// TwinCAT 3 PLC project TcoPneumatics
// Title: TcoPneumatics
// Company: Vortex.Library
// Author: Dustin Hullett
// ProjectVersion: 0.6.0.913
// ProgramVersion: 3.1.4024.12
// libraries:
//   Tc2_Standard, * (Beckhoff Automation GmbH)
//   Tc2_System, * (Beckhoff Automation GmbH)
//   Tc3_Module, * (Beckhoff Automation GmbH)
//   TcoCore, 0.6.0.913 (Vortex.Library)
// project tree:
//   POUs/Cylinders/Base/ TcoCylinderBase.TcPOU, TcoDoubleCylinderBase.TcPOU
//   POUs/Cylinders/ TcoCylinder.TcPOU, TcoCylinderConfig.TcDUT, TcoCylinderStatus.TcDUT, TcoCylinderMoveTask.TcPOU, ITcoCylinder.TcIO, TcoDoubleCylinder.TcPOU
//   Version/ Global_Version.TcGVL
// real-time tasks:
//   TASK PlcTask: cycle T#10ms, priority 20, ADS port 350
//   TASK PlcTask1: cycle T#10ms, priority 21, ADS port 351

// ---- POUs/Cylinders/TcoCylinderConfig.TcDUT
TYPE TcoCylinderConfig :
STRUCT
    TimeToReachHomePosition : TIME := T#10S;
    TimeToReachWorkPosition : TIME := T#10S;
    TimeToRefill : TIME := T#1000MS;
END_STRUCT
END_TYPE

// ---- POUs/Cylinders/TcoCylinderStatus.TcDUT
TYPE TcoCylinderStatus :
STRUCT
    ActionDescription : STRING(100);
END_STRUCT
END_TYPE

// ---- Version/Global_Version.TcGVL
{attribute 'TcGenerated'}
{attribute 'no-analysis'}
{attribute 'linkalways'}
// This function has been automatically generated from the project information.
VAR_GLOBAL CONSTANT
    {attribute 'const_non_replaced'}
    stLibVersion_TcoPneumatics : ST_LibVersion := (
        iMajor := 0,
        iMinor := 1,
        iBuild := 0,
        iRevision := 54,
        nFlags := 0,
        sVersion := '0.1.0.54');
END_VAR

// ---- POUs/Cylinders/ITcoCylinder.TcIO
INTERFACE ITcoCylinder EXTENDS __System.IQueryInterface

PROPERTY AtHome : bool
GET
END_GET
END_PROPERTY

PROPERTY AtWork : bool
GET
END_GET
END_PROPERTY

METHOD MoveToHome : TcoCore.ITcoTaskStatus
END_METHOD

METHOD MoveToWork :TcoCore.ITcoTaskStatus
END_METHOD

(*~
	<docu>
		<summary>
			Stops cyclinder movement.
		 	<remarks>
				<note type="important">
					This method switched off the signals for the movement of the piston in both direction.
					However depending on the pnemumatics configuration the movement may contintue if designed in that way.
					THIS IS NOT A SAFETY FUCTION!
				</note>
			</remarks>
		</summary>
	</docu>
~*)
METHOD Stop : TcoCore.ITcoTaskStatus
END_METHOD

END_INTERFACE

// ---- POUs/Cylinders/Base/TcoCylinderBase.TcPOU
FUNCTION_BLOCK ABSTRACT TcoCylinderBase EXTENDS TcoCore.TcoComponent IMPLEMENTS ITcoCylinder
VAR_IN_OUT
    (*~
        <docu>
            <summary>
                Home position sensor.
            </summary>
        </docu>
    ~*)
    {attribute addProperty Name "<#Home position sensor#>"}
    inoAtHomePos : BOOL;
    (*~
        <docu>
            <summary>
                Working position sensor.
            </summary>
        </docu>
    ~*)
    {attribute addProperty Name "<#Work position sensor#>"}
    inoAtWorkPos : BOOL;
END_VAR
VAR_IN_OUT
    (*~
        <docu>
            <summary>
                Move to working home position signal.
            </summary>
        </docu>
    ~*)
    {attribute addProperty Name "<#Move to home position actuator#>"}
    inoToHomePos : BOOL;
    (*~
        <docu>
            <summary>
                Move to working posistion signal.
            </summary>
        </docu>
    ~*)
    {attribute addProperty Name "<#Move to work position actuator#>"}
    inoToWorkPos : BOOL;
END_VAR
VAR
    (*~
        <docu>
            <summary>
                Home position sensor.
            </summary>
        </docu>
    ~*)
    {attribute addProperty Name "<#Home position sensor#>"}
    _atHomePos : BOOL;
    (*~
        <docu>
            <summary>
                Working position sensor.
            </summary>
        </docu>
    ~*)
    {attribute addProperty Name "<#Work position sensor#>"}
    _atWorkPos : BOOL;
    (*~
        <docu>
            <summary>
                Move to working home position signal.
            </summary>
        </docu>
    ~*)
    {attribute addProperty Name "<#Move to home position actuator#>"}
    _toHomePos : BOOL;
    (*~
        <docu>
            <summary>
                Move to working posistion signal.
            </summary>
        </docu>
    ~*)
    {attribute addProperty Name "<#Move to work position actuator#>"}
    _toWorkPos : BOOL;
END_VAR
VAR
    {attribute addProperty Name "<#Home sensor signal#>"}
    _atHomePosSignalInfo : TcoCore.TcoSignalInfo;
    {attribute addProperty Name "<#Work sensor signal#>"}
    _atWorkPosSignalInfo : TcoCore.TcoSignalInfo;
    {attribute addProperty Name "<#Move to home position signal#>"}
    _toHomePosSignalInfo : TcoCore.TcoSignalInfo;
    {attribute addProperty Name "<#Move to work position signal#>"}
    _toWorkPosSignalInfo : TcoCore.TcoSignalInfo;
END_VAR

IF (__ISVALIDREF(inoAtHomePos)) THEN
    _atHomePos := inoAtHomePos;
    _atHomePosSignalInfo.GetSignalInfo(SIZEOF(inoAtHomePos), ADR(inoAtHomePos));
END_IF;

IF (__ISVALIDREF(inoAtWorkPos)) THEN
    _atWorkPos := inoAtWorkPos;
    _atWorkPosSignalInfo.GetSignalInfo(SIZEOF(inoAtWorkPos), ADR(inoAtWorkPos));
END_IF;

IF (__ISVALIDREF(inoToHomePos)) THEN
    inoToHomePos := _toHomePos;
    _toHomePosSignalInfo.GetSignalInfo(SIZEOF(inoToHomePos), ADR(inoToHomePos));
END_IF;

IF (__ISVALIDREF(inoToWorkPos)) THEN
    inoToWorkPos := _toWorkPos;
    _toWorkPosSignalInfo.GetSignalInfo(SIZEOF(inoToWorkPos), ADR(inoToWorkPos));
END_IF;

(*~
    <docu>
        <summary>
            Gets whether the piston is in home position.
        </summary>
    </docu>
~*)
PROPERTY AtHome : bool
GET
AtHome := THIS^._atHomePos;
END_GET
END_PROPERTY

(*~
    <docu>
        <summary>
            Gets whether the piston is in work position.
        </summary>
    </docu>
~*)
PROPERTY AtWork : bool
GET
AtWork := _atWorkPos;
END_GET
END_PROPERTY

METHOD FB_init : BOOL
VAR_INPUT
    bInitRetains : BOOL; // if TRUE, the retain variables are initialized (warm start / cold start)
    bInCopyCode : BOOL; // if TRUE, the instance afterwards gets moved into the copy code (online change)
    ParentObject : ITcoObject;
END_VAR
END_METHOD

(*~
    <docu>
        <summary>
            Gets the `MoveHomeTask` task that controls the moving of the cyclinder in home position.
            <remarks>
                <note type="important">
                    This is an abstract method and must be implemented in derived class.
                </note>
            </remarks>
        </summary>
    </docu>
~*)
PROPERTY PUBLIC ABSTRACT MoveHomeTask : TcoCore.ITcoTask
GET
END_GET
END_PROPERTY

(*~
    <docu>
        <summary>
            Starts movement into home position.
        </summary>
    </docu>
~*)
METHOD MoveToHome : TcoCore.ITcoTaskStatus
IF (MoveHomeTask <> 0) THEN
    MoveToHome := MoveHomeTask.Invoke();
END_IF;
END_METHOD

(*~
    <docu>
        <summary>
            Starts movement into work position.
        </summary>
    </docu>
~*)
METHOD MoveToWork : TcoCore.ITcoTaskStatus
IF (MoveWorkTask <> 0) THEN
    MoveToWork := MoveWorkTask.Invoke();
END_IF;
END_METHOD

(*~
    <docu>
        <summary>
            Gets the `MoveWorkTask` task that controls the moving of the cyclinder into work position.
            <remarks>
                <note type="important">
                    This is an abstract method and must be implemented in derived class.
                </note>
            </remarks>
        </summary>
    </docu>
~*)
PROPERTY PUBLIC ABSTRACT MoveWorkTask : TcoCore.ITcoTask
GET
END_GET
END_PROPERTY

(*~
    <docu>
        <summary>
            Restore all tasks of this instance into initial state.
        </summary>
    </docu>
~*)
METHOD Restore : ITcoRestorable
IF (MoveHomeTask <> 0) THEN
    MoveHomeTask.Restore();
END_IF;

IF (MoveWorkTask <> 0) THEN
    MoveWorkTask.Restore();
END_IF;

IF (StopTask <> 0) THEN
    StopTask.Restore();
END_IF;
END_METHOD

METHOD PROTECTED ServiceMode
END_METHOD

(*~
    <docu>
        <summary>
            Stops cyclinder movement.
             <remarks>
                <note type="important">
                    This method switched off the signals for the movement of the piston in both direction.
                    However depending on the pnemumatics configuration the movement may contintue if designed in that way.
                    THIS IS NOT A SAFETY FUCTION!
                </note>
            </remarks>
        </summary>
    </docu>
~*)
METHOD Stop : TcoCore.ITcoTaskStatus
IF (StopTask <> 0) THEN
    Stop := StopTask.Invoke();
END_IF;
END_METHOD

(*~
    <docu>
        <summary>
            Gets the `StopTask` task that controls the stopping cyclinder movement.
            <remarks>
                <note type="important">
                    This is an abstract method and must be implemented in derived class.
                </note>
            </remarks>
        </summary>
    </docu>
~*)
PROPERTY PUBLIC ABSTRACT StopTask : TcoCore.ITcoTask
GET
END_GET
END_PROPERTY

END_FUNCTION_BLOCK

// ---- POUs/Cylinders/Base/TcoDoubleCylinderBase.TcPOU
FUNCTION_BLOCK ABSTRACT TcoDoubleCylinderBase EXTENDS TcoCore.TcoComponent IMPLEMENTS ITcoCylinder
VAR_IN_OUT
    (*~
        <docu>
            <summary>
                Home position sensor 1.
            </summary>
        </docu>
    ~*)
    {attribute addProperty Name "<#Home position sensor#> - 1"}
    inoAtHomePos1 : BOOL;
    (*~
        <docu>
            <summary>
                Home position sensor 2.
            </summary>
        </docu>
    ~*)
    {attribute addProperty Name "<#Home position sensor#> - 2"}
    inoAtHomePos2 : BOOL;
    (*~
        <docu>
            <summary>
                Working position sensor 1.
            </summary>
        </docu>
    ~*)
    {attribute addProperty Name "<#Work position sensor#> - 1"}
    inoAtWorkPos1 : BOOL;
    (*~
        <docu>
            <summary>
                Working position sensor 1.
            </summary>
        </docu>
    ~*)
    {attribute addProperty Name "<#Work position sensor#> - 2"}
    inoAtWorkPos2 : BOOL;
END_VAR
VAR_IN_OUT
    (*~
        <docu>
            <summary>
                Move to working home position signal.
            </summary>
        </docu>
    ~*)
    {attribute addProperty Name "<#Move to home position actuator#>"}
    inoToHomePos : BOOL;
    (*~
        <docu>
            <summary>
                Move to working posistion signal.
            </summary>
        </docu>
    ~*)
    {attribute addProperty Name "<#Move to work position actuator#>"}
    inoToWorkPos : BOOL;
END_VAR
VAR
    (*~
        <docu>
            <summary>
                Home position sensor.
            </summary>
        </docu>
    ~*)
    {attribute addProperty Name "<#Home position sensor#>"}
    _atHomePos : BOOL;
    (*~
        <docu>
            <summary>
                Working position sensor.
            </summary>
        </docu>
    ~*)
    {attribute addProperty Name "<#Work position sensor#>"}
    _atWorkPos : BOOL;
    (*~
        <docu>
            <summary>
                Move to working home position signal.
            </summary>
        </docu>
    ~*)
    {attribute addProperty Name "<#Move to home position actuator#>"}
    _toHomePos : BOOL;
    (*~
        <docu>
            <summary>
                Move to working posistion signal.
            </summary>
        </docu>
    ~*)
    {attribute addProperty Name "<#Move to work position actuator#>"}
    _toWorkPos : BOOL;
END_VAR
VAR
    {attribute addProperty Name "<#Home sensor signal 1#>"}
    _atHomePos1SignalInfo : TcoCore.TcoSignalInfo;
    {attribute addProperty Name "<#Home sensor signal 2#>"}
    _atHomePos2SignalInfo : TcoCore.TcoSignalInfo;
    {attribute addProperty Name "<#Work sensor signal 1#>"}
    _atWorkPos1SignalInfo : TcoCore.TcoSignalInfo;
    {attribute addProperty Name "<#Work sensor signal 2#>"}
    _atWorkPos2SignalInfo : TcoCore.TcoSignalInfo;
    {attribute addProperty Name "<#Move to home position signal#>"}
    _toHomePosSignalInfo : TcoCore.TcoSignalInfo;
    {attribute addProperty Name "<#Move to work position signal#>"}
    _toWorkPosSignalInfo : TcoCore.TcoSignalInfo;
END_VAR

IF (__ISVALIDREF(inoAtHomePos1) AND __ISVALIDREF(inoAtHomePos2)) THEN
    _atHomePos := inoAtHomePos1 AND inoAtHomePos2;
    _atHomePos1SignalInfo.GetSignalInfo(SIZEOF(inoAtHomePos1), ADR(inoAtHomePos1));
    _atHomePos2SignalInfo.GetSignalInfo(SIZEOF(inoAtHomePos2), ADR(inoAtHomePos2));
END_IF;

IF (__ISVALIDREF(inoAtWorkPos1) AND __ISVALIDREF(inoAtWorkPos2)) THEN
    _atWorkPos := inoAtWorkPos1 AND inoAtWorkPos2;
    _atWorkPos1SignalInfo.GetSignalInfo(SIZEOF(inoAtWorkPos1), ADR(inoAtWorkPos1));
    _atWorkPos2SignalInfo.GetSignalInfo(SIZEOF(inoAtWorkPos2), ADR(inoAtWorkPos2));
END_IF;

IF (__ISVALIDREF(inoToHomePos)) THEN
    inoToHomePos := _toHomePos;
    _toHomePosSignalInfo.GetSignalInfo(SIZEOF(inoToHomePos), ADR(inoToHomePos));
END_IF;

IF (__ISVALIDREF(inoToWorkPos)) THEN
    inoToWorkPos := _toWorkPos;
    _toWorkPosSignalInfo.GetSignalInfo(SIZEOF(inoToWorkPos), ADR(inoToWorkPos));
END_IF;

(*~
    <docu>
        <summary>
            Gets whether the piston is in home position.
        </summary>
    </docu>
~*)
PROPERTY AtHome : bool
GET
AtHome := THIS^._atHomePos;
END_GET
END_PROPERTY

(*~
    <docu>
        <summary>
            Gets whether the piston is in work position.
        </summary>
    </docu>
~*)
PROPERTY AtWork : bool
GET
AtWork := _atWorkPos;
END_GET
END_PROPERTY

METHOD FB_init : BOOL
VAR_INPUT
    bInitRetains : BOOL; // if TRUE, the retain variables are initialized (warm start / cold start)
    bInCopyCode : BOOL; // if TRUE, the instance afterwards gets moved into the copy code (online change)
    ParentObject : ITcoObject;
END_VAR
END_METHOD

(*~
    <docu>
        <summary>
            Gets the `MoveHomeTask` task that controls the moving of the cyclinder in home position.
            <remarks>
                <note type="important">
                    This is an abstract method and must be implemented in derived class.
                </note>
            </remarks>
        </summary>
    </docu>
~*)
PROPERTY PUBLIC ABSTRACT MoveHomeTask : TcoCore.ITcoTask
GET
END_GET
END_PROPERTY

(*~
    <docu>
        <summary>
            Starts movement into home position.
        </summary>
    </docu>
~*)
METHOD MoveToHome : TcoCore.ITcoTaskStatus
IF (MoveHomeTask <> 0) THEN
    MoveToHome := MoveHomeTask.Invoke();
END_IF;
END_METHOD

(*~
    <docu>
        <summary>
            Starts movement into work position.
        </summary>
    </docu>
~*)
METHOD MoveToWork : TcoCore.ITcoTaskStatus
IF (MoveWorkTask <> 0) THEN
    MoveToWork := MoveWorkTask.Invoke();
END_IF;
END_METHOD

(*~
    <docu>
        <summary>
            Gets the `MoveWorkTask` task that controls the moving of the cyclinder into work position.
            <remarks>
                <note type="important">
                    This is an abstract method and must be implemented in derived class.
                </note>
            </remarks>
        </summary>
    </docu>
~*)
PROPERTY PUBLIC ABSTRACT MoveWorkTask : TcoCore.ITcoTask
GET
END_GET
END_PROPERTY

(*~
    <docu>
        <summary>
            Restore all tasks of this instance into initial state.
        </summary>
    </docu>
~*)
METHOD Restore : ITcoRestorable
IF (MoveHomeTask <> 0) THEN
    MoveHomeTask.Restore();
END_IF;

IF (MoveWorkTask <> 0) THEN
    MoveWorkTask.Restore();
END_IF;

IF (StopTask <> 0) THEN
    StopTask.Restore();
END_IF;
END_METHOD

METHOD PROTECTED ServiceMode
END_METHOD

(*~
    <docu>
        <summary>
            Stops cyclinder movement.
             <remarks>
                <note type="important">
                    This method switched off the signals for the movement of the piston in both direction.
                    However depending on the pnemumatics configuration the movement may contintue if designed in that way.
                    THIS IS NOT A SAFETY FUCTION!
                </note>
            </remarks>
        </summary>
    </docu>
~*)
METHOD Stop : TcoCore.ITcoTaskStatus
IF (StopTask <> 0) THEN
    Stop := StopTask.Invoke();
END_IF;
END_METHOD

(*~
    <docu>
        <summary>
            Gets the `StopTask` task that controls the stopping cyclinder movement.
            <remarks>
                <note type="important">
                    This is an abstract method and must be implemented in derived class.
                </note>
            </remarks>
        </summary>
    </docu>
~*)
PROPERTY PUBLIC ABSTRACT StopTask : TcoCore.ITcoTask
GET
END_GET
END_PROPERTY

END_FUNCTION_BLOCK

// ---- POUs/Cylinders/TcoCylinder.TcPOU
{attribute addProperty _moveHomeDefaultName "<#MOVE HOME#>"}
{attribute addProperty _moveWorkDefaultName "<#MOVE TO WORK#>"}
{attribute addProperty _stopDefaultName "<#STOP#>"}
FUNCTION_BLOCK TcoCylinder EXTENDS TcoCylinderBase
VAR
    {attribute addProperty Name "|[[1]Attribute_moveHomeDefaultName]|"}
    _moveHomeDefault : TcoCylinderMoveTask(THIS^);
    {attribute addProperty Name "|[[1]Attribute_moveWorkDefaultName]|"}
    _moveWorkDefault : TcoCylinderMoveTask(THIS^);
    {attribute addProperty Name "|[[1]Attribute_stopDefaultName]|"}
    _stopDefault : TcoCore.TcoTask(THIS^);
	increment: INT;
	_suspendedHome:BOOL;
	_suspendedWork:BOOL;
	{attribute 'hide'} 
	_suspendedHomeCounter:INT;
	{attribute 'hide'} 
	_suspendedWorkCounter:INT;
END_VAR
VAR
    _config : TcoCylinderConfig;
	_status : TcoCylinderStatus;
	_refillTimer:TON;	
END_VAR

SUPER^(inoAtHomePos := inoAtHomePos, inoAtWorkPos := inoAtWorkPos, inoToHomePos := inoToHomePos, inoToWorkPos := inoToWorkPos);
_suspendedHomeCounter:=0;
_suspendedWorkCounter:=0;

	
IF(_atHomePos AND _atWorkPos) THEN Messenger.Error('<#Home and work position sensors are both active. Check the position of sensors!#>'); END_IF;

// Disables mutualy exclusive actions
_moveWorkDefault.Enabled := TRUE;// NOT _moveHomeDefault.Busy;


_moveHomeDefault(PositionSensor := _atHomePos AND NOT _atWorkPos,
    MoveToPositionSignal := _toHomePos,
    InverseSignal := _toWorkPos,
	TimeToRefill:=_config.TimeToRefill,
	refInverseTask:=_moveWorkDefault,
    MaxTimeToReachPosition := _config.TimeToReachHomePosition,
    PositionName := '<#Home#>');


	
// Disables mutualy exclusive actions		
_moveHomeDefault.Enabled := TRUE;//NOT _moveWorkDefault.Busy;
	
_moveWorkDefault(PositionSensor := _atWorkPos AND NOT _atHomePos,
    MoveToPositionSignal := _toWorkPos,
    InverseSignal := _toHomePos,
	TimeToRefill:=_config.TimeToRefill,
	refInverseTask:=_moveHomeDefault,
    MaxTimeToReachPosition := _config.TimeToReachWorkPosition,
    PositionName := '<#Work#>');
	

IF (_stopDefault.Execute()) THEN
	_toHomePos := FALSE;
	_toWorkPos := FALSE;
    _moveHomeDefault.Abort();
    _moveWorkDefault.Abort();
    _stopDefault.Abort();
    _moveHomeDefault.Restore();
    _moveWorkDefault.Restore();
    _stopDefault.Restore();
    _stopDefault.DoneWhen(TRUE);
END_IF



// For further discussion about Status
IF(_moveHomeDefault.Busy) THEN
	_status.ActionDescription := 'Moving to home position';
ELSIF(_moveWorkDefault.Busy) THEN
	_status.ActionDescription := 'Moving to work position';
ELSIF(_stopDefault.Busy) THEN
	_status.ActionDescription := 'Stopping pressure';
ELSE	
	_status.ActionDescription := 'Idle';
END_IF

SUPER^(inoAtHomePos := inoAtHomePos, inoAtWorkPos := inoAtWorkPos, inoToHomePos := inoToHomePos, inoToWorkPos := inoToWorkPos);

(*~
	<docu>
		<summary>
			Aborts the movement to home position when the condition is 'true'.
		</summary>
		<remarks>			
				<note type="warning">
					The call of this method will be effective only when called AFTER the initialization of the instance of given TcoCylinder.
				</note>
		</remarks>	
	</docu>
~*)
METHOD AbortMoveHome : BOOL
VAR_IN_OUT
	(*~
	<docu>
		<summary>
			Condition to abort the movement of the cylinder.
		</summary>	
	</docu>
	~*)
	inoDisableCondition : BOOL;
END_VAR
VAR
	_signalInfo : TcoSignalInfo;
END_VAR
IF (_toHomePos OR _moveHomeDefault.Busy) AND inoDisableCondition THEN
	_signalInfo.GetSignalInfo(SIZEOF(inoDisableCondition), ADR(inoDisableCondition));
	Messenger.Build().Append('<#Movement aborted due to#> : ').Append(_signalInfo.SymbolPath).As().AsError().Pin();
	_toHomePos := FALSE;
	IF(__ISVALIDREF(THIS^.inoToHomePos)) THEN THIS^.inoToHomePos := FALSE; END_IF;
	_moveHomeDefault.Abort();
END_IF
END_METHOD

(*~
	<docu>
		<summary>
			Aborts the movement to work position when the condition is 'true'.
		</summary>
		<remarks>			
				<note type="warning">
					The call of this method will be effective only when called AFTER the initialization of the instance of given TcoCylinder.
				</note>
		</remarks>	
	</docu>
~*)
METHOD AbortMoveWork : BOOL
VAR_IN_OUT
	(*~
		<docu>
			<summary>
				Condition to abort the movement of the cylinder.
			</summary>	
		</docu>
	~*)
	inoDisableCondition : BOOL;
END_VAR
VAR
	_signalInfo : TcoSignalInfo;
END_VAR
IF (_toWorkPos OR _moveWorkDefault.Busy) AND inoDisableCondition THEN
	_signalInfo.GetSignalInfo(SIZEOF(inoDisableCondition), ADR(inoDisableCondition));
	Messenger.Build().Append('<#Movement aborted due to#> : ').Append(_signalInfo.SymbolPath).As().AsError().Pin();
	_toWorkPos := FALSE;
	IF(__ISVALIDREF(THIS^.inoToWorkPos)) THEN THIS^.inoToWorkPos := FALSE; END_IF;
	_moveWorkDefault.Abort();
END_IF
END_METHOD

(*~
	<docu>
		<summary>
			Gets the configuration of the cylinder. 					
		</summary>			
	</docu>	
~*)
PROPERTY Config : REFERENCE TO TcoCylinderConfig
GET
Config REF= _config;
END_GET
END_PROPERTY

(*~
	<docu>
		<summary>
			Gets the `MoveHomeTask` task that controls the moving of the cyclinder in home position. 		
		</summary>			
	</docu>	
~*)
PROPERTY MoveHomeTask : TcoCore.ITcoTask
GET
MoveHomeTask := _moveHomeDefault;
END_GET
END_PROPERTY

(*~
	<docu>
		<summary>
			Gets the `MoveWorkTask` task that controls the moving of the cyclinder into work position. 		
		</summary>			
	</docu>	
~*)
PROPERTY MoveWorkTask : TcoCore.ITcoTask
GET
MoveWorkTask := _moveWorkDefault;
END_GET
END_PROPERTY

(*~
	<docu>
		<summary>
			Refill cylinder after booth outputs are off .
		</summary>
		<remarks>			
				<note type="warning">
					The call of this method will be effective only when called AFTER the initialization of the instance of given TcoCylinder and methods like AbortMoveHone,SuspendMoveHom...
				</note>
		</remarks>	
	</docu>
~*)
METHOD Refill : BOOL
VAR_INPUT
	(*~
	<docu>
		<summary>
			Time of refill cylinder after aborting or suspending
		</summary>	
	</docu>
	~*)
	inRefillTime:TIME;
END_VAR

_refillTimer(In:=inoToHomePos XOR  inoToWorkPos ,Pt:=T#49D);

_config.TimeToRefill:=inRefillTime;

IF  _refillTimer.ET>T#0MS
	AND _refillTimer.ET<_config.TimeToRefill  
	AND _config.TimeToRefill<>T#0S THEN
	_toHomePos	 := TRUE;
	_toWorkPos	 := TRUE;	
END_IF;

	
SUPER^(inoAtHomePos := inoAtHomePos, inoAtWorkPos := inoAtWorkPos, inoToHomePos := inoToHomePos, inoToWorkPos := inoToWorkPos);
END_METHOD

PROPERTY Status : REFERENCE TO TcoCylinderStatus
GET
Status REF= _status;
END_GET
END_PROPERTY

(*~
	<docu>
		<summary>
			Gets the `StopTask` task that controls the stopping of the cyclinder. 		
		</summary>			
	</docu>	
~*)
PROPERTY StopTask : TcoCore.ITcoTask
GET
StopTask := _stopDefault;
END_GET
END_PROPERTY

(*~
	<docu>
		<summary>
			Suspend the movement to home position when the condition is 'true'. Task is still busy
		</summary>
		<remarks>			
				<note type="warning">
					The call of this method will be effective only when called AFTER the initialization of the instance of given TcoCylinder.
				</note>
		</remarks>	
	</docu>
~*)
METHOD SuspendMoveHome : BOOL
VAR_IN_OUT
	(*~
	<docu>
		<summary>
			Condition to abort the movement of the cylinder.
		</summary>	
	</docu>
	~*)
	inoDisableCondition : BOOL;
END_VAR
VAR
	_signalInfo : TcoSignalInfo;
END_VAR
IF inoDisableCondition THEN
	_suspendedHomeCounter:=_suspendedHomeCounter+1;
END_IF
_suspendedHome:=_suspendedHomeCounter>0;

IF (_toHomePos OR _moveHomeDefault.Busy) AND inoDisableCondition THEN
	_signalInfo.GetSignalInfo(SIZEOF(inoDisableCondition), ADR(inoDisableCondition));
	Messenger.Warning(CONCAT('<#Movement suspended due to#> : ' , _signalInfo.SymbolPath));
	_toHomePos := FALSE;
	IF(__ISVALIDREF(THIS^.inoToHomePos)) THEN THIS^.inoToHomePos := FALSE; END_IF;
	
END_IF
END_METHOD

METHOD SuspendMoveHomeExpression : BOOL
VAR_INPUT
		inDisableCondition : BOOL;
		inMessage:STRING;
END_VAR
IF inDisableCondition THEN
	_suspendedHomeCounter:=_suspendedHomeCounter+1;
END_IF
_suspendedHome:=_suspendedHomeCounter>0;

IF (_toHomePos OR _moveHomeDefault.Busy) AND inDisableCondition THEN
	Messenger.Warning(CONCAT('<#Movement suspended due to#> : ' , inMessage));
	_toHomePos := FALSE;
	IF(__ISVALIDREF(THIS^.inoToHomePos)) THEN THIS^.inoToHomePos := FALSE; END_IF;
	
END_IF;
END_METHOD

(*~
	<docu>
		<summary>
			Suspend the movement to home position when the condition is NOT 'true'. Task is still busy
		</summary>
		<remarks>			
				<note type="warning">
					The call of this method will be effective only when called AFTER the initialization of the instance of given TcoCylinder.
				</note>
		</remarks>	
	</docu>
~*)
METHOD SuspendMoveHomeInverted : BOOL
VAR_IN_OUT
	(*~
	<docu>
		<summary>
			Condition to abort the movement of the cylinder.
		</summary>	
	</docu>
	~*)
	inoDisableCondition : BOOL;
END_VAR
VAR
	_signalInfo : TcoSignalInfo;
END_VAR
IF inoDisableCondition THEN
	_suspendedHomeCounter:=_suspendedHomeCounter+1;
END_IF
_suspendedHome:=_suspendedHomeCounter>0;

IF (_toHomePos OR _moveHomeDefault.Busy) AND not inoDisableCondition THEN
	_signalInfo.GetSignalInfo(SIZEOF(inoDisableCondition), ADR(inoDisableCondition));
	Messenger.Warning(CONCAT('<#Movement suspended due to NOT#> : ' , _signalInfo.SymbolPath));
	_toHomePos := FALSE;
	IF(__ISVALIDREF(THIS^.inoToHomePos)) THEN THIS^.inoToHomePos := FALSE; END_IF;
	
END_IF
END_METHOD

(*~
	<docu>
		<summary>
			Suspend the movement to work position when the condition is 'true'. Task is still bussy
		</summary>
		<remarks>			
				<note type="warning">
					The call of this method will be effective only when called AFTER the initialization of the instance of given TcoCylinder.
				</note>
		</remarks>	
	</docu>
~*)
METHOD SuspendMoveWork : BOOL
VAR_IN_OUT
	(*~
		<docu>
			<summary>
				Condition to abort the movement of the cylinder.
			</summary>	
		</docu>
	~*)
	inoDisableCondition : BOOL;
END_VAR
VAR
	_signalInfo : TcoSignalInfo;
END_VAR
IF inoDisableCondition THEN
	_suspendedWorkCounter:=_suspendedWorkCounter+1;
END_IF
_suspendedWork:=_suspendedWorkCounter>0;

IF (_toWorkPos OR _moveWorkDefault.Busy) AND inoDisableCondition THEN
	_signalInfo.GetSignalInfo(SIZEOF(inoDisableCondition), ADR(inoDisableCondition));
	Messenger.Warning(CONCAT('<#Movement suspended due to#> : ' , _signalInfo.SymbolPath));
	_toWorkPos := FALSE;
	IF(__ISVALIDREF(THIS^.inoToWorkPos)) THEN THIS^.inoToWorkPos := FALSE; END_IF;

END_IF
END_METHOD

METHOD SuspendMoveWorkExpression : BOOL
VAR_INPUT
		inDisableCondition : BOOL;
		inMessage:STRING;
END_VAR
IF inDisableCondition THEN
	_suspendedWorkCounter:=_suspendedWorkCounter+1;
END_IF
_suspendedWork:=_suspendedWorkCounter>0;

IF (_toWorkPos OR _moveWorkDefault.Busy) AND inDisableCondition THEN
    Messenger.Warning(CONCAT('<#Movement suspended due to#> : ', inMessage));
    _toWorkPos := FALSE;
    IF (__ISVALIDREF(THIS^.inoToWorkPos)) THEN
        THIS^.inoToWorkPos := FALSE;
    END_IF;

END_IF
END_METHOD

(*~
	<docu>
		<summary>
			Suspend the movement to work position when the condition is NOT 'true'. Task is still busy
		</summary>
		<remarks>			
				<note type="warning">
					The call of this method will be effective only when called AFTER the initialization of the instance of given TcoCylinder.
				</note>
		</remarks>	
	</docu>
~*)
METHOD SuspendMoveWorkInverted : BOOL
VAR_IN_OUT
	(*~
		<docu>
			<summary>
				Condition to abort the movement of the cylinder.
			</summary>	
		</docu>
	~*)
	inoDisableCondition : BOOL;
END_VAR
VAR
	_signalInfo : TcoSignalInfo;
END_VAR
IF inoDisableCondition THEN
	_suspendedWorkCounter:=_suspendedWorkCounter+1;
END_IF
_suspendedWork:=_suspendedWorkCounter>0;

IF (_toWorkPos OR _moveWorkDefault.Busy) AND not inoDisableCondition THEN
    _signalInfo.GetSignalInfo(SIZEOF(inoDisableCondition), ADR(inoDisableCondition));
    Messenger.Warning(CONCAT('<#Movement suspended due to NOT#> : ', _signalInfo.SymbolPath));
    _toWorkPos := FALSE;
    IF (__ISVALIDREF(THIS^.inoToWorkPos)) THEN
        THIS^.inoToWorkPos := FALSE;
    END_IF;

END_IF
END_METHOD

END_FUNCTION_BLOCK

// ---- POUs/Cylinders/TcoCylinderMoveTask.TcPOU
FUNCTION_BLOCK TcoCylinderMoveTask EXTENDS TcoCore.TcoTask
VAR_INPUT
    PositionSensor : BOOL;
    MaxTimeToReachPosition : TIME := T#10S;
    TimeToRefill : TIME := T#100MS;
    PositionName : STRING(25);
END_VAR
VAR_IN_OUT
    MoveToPositionSignal : BOOL;
    InverseSignal : BOOL;
END_VAR
VAR
    _stringBuilder : TcoCore.StringBuilder;
END_VAR

IF (THIS^.Execute()) THEN
    IF (THIS^.ElapsedTime > MaxTimeToReachPosition) THEN
        THIS^.Messenger.Warning(_stringBuilder.Clear().Append(PositionName).Append(' sensor not reached yet.').ToString());
    END_IF;

    InverseSignal := FALSE;
    MoveToPositionSignal := TRUE;
    THIS^.DoneWhen(PositionSensor);
END_IF

METHOD PUBLIC FB_init : BOOL
VAR_INPUT
    bInitRetains : BOOL; // if TRUE, the retain variables are initialized (warm start / cold start)
    bInCopyCode : BOOL; // if TRUE, the instance afterwards gets moved into the copy code (online change)
    ParentObject : ITcoObject;
END_VAR
END_METHOD

(*~
    <docu>
        <summary>
            Executes when task is aborted.
        </summary>
    </docu>
~*)
METHOD PROTECTED OnAbort
MoveToPositionSignal := FALSE;
END_METHOD

METHOD PROTECTED OnError
END_METHOD

METHOD PROTECTED OnStart
END_METHOD

END_FUNCTION_BLOCK

// ---- POUs/Cylinders/TcoDoubleCylinder.TcPOU
{attribute addProperty _moveHomeDefaultName "<#MOVE HOME#>"}
{attribute addProperty _moveWorkDefaultName "<#MOVE TO WORK#>"}
{attribute addProperty _stopDefaultName "<#STOP#>"}
FUNCTION_BLOCK TcoDoubleCylinder EXTENDS TcoDoubleCylinderBase
VAR
    {attribute addProperty Name "|[[1]Attribute_moveHomeDefaultName]|"}
    _moveHomeDefault : TcoCylinderMoveTask(THIS^);
    {attribute addProperty Name "|[[1]Attribute_moveWorkDefaultName]|"}
    _moveWorkDefault : TcoCylinderMoveTask(THIS^);
    {attribute addProperty Name "|[[1]Attribute_stopDefaultName]|"}
    _stopDefault : TcoCore.TcoTask(THIS^);
    increment : INT;
END_VAR
VAR
    _config : TcoCylinderConfig;
    _status : TcoCylinderStatus;
    _refillTimer : TON;
END_VAR

SUPER^(inoAtHomePos1 := inoAtHomePos1,
    inoAtHomePos2 := inoAtHomePos2,
    inoAtWorkPos1 := inoAtWorkPos1,
    inoAtWorkPos2 := inoAtWorkPos2,
    inoToHomePos := inoToHomePos,
    inoToWorkPos := inoToWorkPos);

IF (_atHomePos AND _atWorkPos) THEN
    Messenger.Error('<#Home and work position sensors are both active. Check the position of sensors!#>');
END_IF;
// Disables mutualy exclusive actions
_moveWorkDefault.Enabled := TRUE; // NOT _moveHomeDefault.Busy;

_moveHomeDefault(PositionSensor := _atHomePos AND NOT _atWorkPos,
    MoveToPositionSignal := _toHomePos,
    InverseSignal := _toWorkPos,
    TimeToRefill := _config.TimeToRefill,
    MaxTimeToReachPosition := _config.TimeToReachHomePosition,
    PositionName := '<#Home#>');

IF _moveHomeDefault.Execute() THEN
    _moveWorkDefault.Restore();
END_IF
// Disables mutualy exclusive actions
_moveHomeDefault.Enabled := true; // NOT _moveWorkDefault.Busy;

_moveWorkDefault(PositionSensor := _atWorkPos AND NOT _atHomePos,
    MoveToPositionSignal := _toWorkPos,
    InverseSignal := _toHomePos,
    TimeToRefill := _config.TimeToRefill,
    MaxTimeToReachPosition := _config.TimeToReachWorkPosition,
    PositionName := '<#Work#>');

IF _moveWorkDefault.Execute() THEN
    _moveHomeDefault.Restore();
END_IF

IF (_stopDefault.Execute()) THEN
    _toHomePos := FALSE;
    _toWorkPos := FALSE;
    _moveHomeDefault.Abort();
    _moveWorkDefault.Abort();
    _stopDefault.Abort();
    _moveHomeDefault.Restore();
    _moveWorkDefault.Restore();
    _stopDefault.Restore();
    _stopDefault.DoneWhen(TRUE);
END_IF

// For further discussion about Status
IF (_moveHomeDefault.Busy) THEN
    _status.ActionDescription := 'Moving to home position';
ELSIF (_moveWorkDefault.Busy) THEN
    _status.ActionDescription := 'Moving to work position';
ELSIF (_stopDefault.Busy) THEN
    _status.ActionDescription := 'Stopping pressure';
ELSE
    _status.ActionDescription := 'Idle';
END_IF

SUPER^(inoAtHomePos1 := inoAtHomePos1,
    inoAtHomePos2 := inoAtHomePos2,
    inoAtWorkPos1 := inoAtWorkPos1,
    inoAtWorkPos2 := inoAtWorkPos2,
    inoToHomePos := inoToHomePos,
    inoToWorkPos := inoToWorkPos);

(*~
    <docu>
        <summary>
            Aborts the movement to home position when the condition is 'true'.
        </summary>
        <remarks>
                <note type="warning">
                    The call of this method will be effective only when called AFTER the initialization of the instance of given TcoCylinder.
                </note>
        </remarks>
    </docu>
~*)
METHOD AbortMoveHome : BOOL
VAR_IN_OUT
    (*~
    <docu>
        <summary>
            Condition to abort the movement of the cylinder.
        </summary>
    </docu>
    ~*)
    inoDisableCondition : BOOL;
END_VAR
VAR
    _signalInfo : TcoSignalInfo;
END_VAR
IF (_toHomePos OR _moveHomeDefault.Busy) AND inoDisableCondition THEN
    _signalInfo.GetSignalInfo(SIZEOF(inoDisableCondition), ADR(inoDisableCondition));
    Messenger.Build().Append('<#Movement aborted due to#> : ').Append(_signalInfo.SymbolPath).As().AsError().Pin();
    _toHomePos := FALSE;

    IF (__ISVALIDREF(THIS^.inoToHomePos)) THEN
        THIS^.inoToHomePos := FALSE;
    END_IF;

    _moveHomeDefault.Abort();
END_IF
END_METHOD

(*~
    <docu>
        <summary>
            Aborts the movement to work position when the condition is 'true'.
        </summary>
        <remarks>
                <note type="warning">
                    The call of this method will be effective only when called AFTER the initialization of the instance of given TcoCylinder.
                </note>
        </remarks>
    </docu>
~*)
METHOD AbortMoveWork : BOOL
VAR_IN_OUT
    (*~
        <docu>
            <summary>
                Condition to abort the movement of the cylinder.
            </summary>
        </docu>
    ~*)
    inoDisableCondition : BOOL;
END_VAR
VAR
    _signalInfo : TcoSignalInfo;
END_VAR
IF (_toWorkPos OR _moveWorkDefault.Busy) AND inoDisableCondition THEN
    _signalInfo.GetSignalInfo(SIZEOF(inoDisableCondition), ADR(inoDisableCondition));
    Messenger.Build().Append('<#Movement aborted due to#> : ').Append(_signalInfo.SymbolPath).As().AsError().Pin();
    _toWorkPos := FALSE;

    IF (__ISVALIDREF(THIS^.inoToWorkPos)) THEN
        THIS^.inoToWorkPos := FALSE;
    END_IF;

    _moveWorkDefault.Abort();
END_IF
END_METHOD

(*~
    <docu>
        <summary>
            Gets the configuration of the cylinder.
        </summary>
    </docu>
~*)
PROPERTY Config : REFERENCE TO TcoCylinderConfig
GET
Config REF= _config;
END_GET
END_PROPERTY

(*~
    <docu>
        <summary>
            Gets the `MoveHomeTask` task that controls the moving of the cyclinder in home position.
        </summary>
    </docu>
~*)
PROPERTY MoveHomeTask : TcoCore.ITcoTask
GET
MoveHomeTask := _moveHomeDefault;
END_GET
END_PROPERTY

(*~
    <docu>
        <summary>
            Gets the `MoveWorkTask` task that controls the moving of the cyclinder into work position.
        </summary>
    </docu>
~*)
PROPERTY MoveWorkTask : TcoCore.ITcoTask
GET
MoveWorkTask := _moveWorkDefault;
END_GET
END_PROPERTY

(*~
    <docu>
        <summary>
            Refill cylinder after booth outputs are off .
        </summary>
        <remarks>
                <note type="warning">
                    The call of this method will be effective only when called AFTER the initialization of the instance of given TcoCylinder and methods like AbortMoveHone,SuspendMoveHom...
                </note>
        </remarks>
    </docu>
~*)
METHOD Refill : BOOL
VAR_INPUT
    (*~
    <docu>
        <summary>
            Time of refill cylinder after aborting or suspending
        </summary>
    </docu>
    ~*)
    inRefillTime : TIME;
END_VAR
_refillTimer(In := inoToHomePos XOR inoToWorkPos, Pt := T#49D);
_config.TimeToRefill := inRefillTime;

IF _refillTimer.ET > T#0MS AND _refillTimer.ET < _config.TimeToRefill AND _config.TimeToRefill <> T#0S THEN
    _toHomePos := TRUE;
    _toWorkPos := TRUE;
END_IF;

SUPER^(inoAtHomePos1 := inoAtHomePos1,
    inoAtHomePos2 := inoAtHomePos2,
    inoAtWorkPos1 := inoAtWorkPos1,
    inoAtWorkPos2 := inoAtWorkPos2,
    inoToHomePos := inoToHomePos,
    inoToWorkPos := inoToWorkPos);
END_METHOD

PROPERTY Status : REFERENCE TO TcoCylinderStatus
GET
Status REF= _status;
END_GET
END_PROPERTY

(*~
    <docu>
        <summary>
            Gets the `StopTask` task that controls the stopping of the cyclinder.
        </summary>
    </docu>
~*)
PROPERTY StopTask : TcoCore.ITcoTask
GET
StopTask := _stopDefault;
END_GET
END_PROPERTY

(*~
    <docu>
        <summary>
            Suspend the movement to home position when the condition is 'true'. Task is still busy
        </summary>
        <remarks>
                <note type="warning">
                    The call of this method will be effective only when called AFTER the initialization of the instance of given TcoCylinder.
                </note>
        </remarks>
    </docu>
~*)
METHOD SuspendMoveHome : BOOL
VAR_IN_OUT
    (*~
    <docu>
        <summary>
            Condition to abort the movement of the cylinder.
        </summary>
    </docu>
    ~*)
    inoDisableCondition : BOOL;
END_VAR
VAR
    _signalInfo : TcoSignalInfo;
END_VAR
IF (_toHomePos OR _moveHomeDefault.Busy) AND inoDisableCondition THEN
    _signalInfo.GetSignalInfo(SIZEOF(inoDisableCondition), ADR(inoDisableCondition));
    Messenger.Warning(CONCAT('<#Movement suspended due to#> : ', _signalInfo.SymbolPath));
    _toHomePos := FALSE;

    IF (__ISVALIDREF(THIS^.inoToHomePos)) THEN
        THIS^.inoToHomePos := FALSE;
    END_IF;
END_IF
END_METHOD

METHOD SuspendMoveHomeExpression : BOOL
VAR_INPUT
    inDisableCondition : BOOL;
    inMessage : STRING;
END_VAR
IF (_toHomePos OR _moveHomeDefault.Busy) AND inDisableCondition THEN
    Messenger.Warning(CONCAT('<#Movement suspended due to#> : ', inMessage));
    _toHomePos := FALSE;

    IF (__ISVALIDREF(THIS^.inoToHomePos)) THEN
        THIS^.inoToHomePos := FALSE;
    END_IF;
END_IF;
END_METHOD

(*~
    <docu>
        <summary>
            Suspend the movement to home position when the condition is NOT 'true'. Task is still busy
        </summary>
        <remarks>
                <note type="warning">
                    The call of this method will be effective only when called AFTER the initialization of the instance of given TcoCylinder.
                </note>
        </remarks>
    </docu>
~*)
METHOD SuspendMoveHomeInverted : BOOL
VAR_IN_OUT
    (*~
    <docu>
        <summary>
            Condition to abort the movement of the cylinder.
        </summary>
    </docu>
    ~*)
    inoDisableCondition : BOOL;
END_VAR
VAR
    _signalInfo : TcoSignalInfo;
END_VAR
IF (_toHomePos OR _moveHomeDefault.Busy) AND NOT inoDisableCondition THEN
    _signalInfo.GetSignalInfo(SIZEOF(inoDisableCondition), ADR(inoDisableCondition));
    Messenger.Warning(CONCAT('<#Movement suspended due to NOT#> : ', _signalInfo.SymbolPath));
    _toHomePos := FALSE;

    IF (__ISVALIDREF(THIS^.inoToHomePos)) THEN
        THIS^.inoToHomePos := FALSE;
    END_IF;
END_IF
END_METHOD

(*~
    <docu>
        <summary>
            Suspend the movement to work position when the condition is 'true'. Task is still bussy
        </summary>
        <remarks>
                <note type="warning">
                    The call of this method will be effective only when called AFTER the initialization of the instance of given TcoCylinder.
                </note>
        </remarks>
    </docu>
~*)
METHOD SuspendMoveWork : BOOL
VAR_IN_OUT
    (*~
        <docu>
            <summary>
                Condition to abort the movement of the cylinder.
            </summary>
        </docu>
    ~*)
    inoDisableCondition : BOOL;
END_VAR
VAR
    _signalInfo : TcoSignalInfo;
END_VAR
IF (_toWorkPos OR _moveWorkDefault.Busy) AND inoDisableCondition THEN
    _signalInfo.GetSignalInfo(SIZEOF(inoDisableCondition), ADR(inoDisableCondition));
    Messenger.Warning(CONCAT('<#Movement suspended due to#> : ', _signalInfo.SymbolPath));
    _toWorkPos := FALSE;

    IF (__ISVALIDREF(THIS^.inoToWorkPos)) THEN
        THIS^.inoToWorkPos := FALSE;
    END_IF;
END_IF
END_METHOD

METHOD SuspendMoveWorkExpression : BOOL
VAR_INPUT
    inDisableCondition : BOOL;
    inMessage : STRING;
END_VAR
IF (_toWorkPos OR _moveWorkDefault.Busy) AND inDisableCondition THEN
    Messenger.Warning(CONCAT('<#Movement suspended due to#> : ', inMessage));
    _toWorkPos := FALSE;

    IF (__ISVALIDREF(THIS^.inoToWorkPos)) THEN
        THIS^.inoToWorkPos := FALSE;
    END_IF;
END_IF
END_METHOD

(*~
    <docu>
        <summary>
            Suspend the movement to work position when the condition is NOT 'true'. Task is still bussy
        </summary>
        <remarks>
                <note type="warning">
                    The call of this method will be effective only when called AFTER the initialization of the instance of given TcoCylinder.
                </note>
        </remarks>
    </docu>
~*)
METHOD SuspendMoveWorkInverted : BOOL
VAR_IN_OUT
    (*~
        <docu>
            <summary>
                Condition to abort the movement of the cylinder.
            </summary>
        </docu>
    ~*)
    inoDisableCondition : BOOL;
END_VAR
VAR
    _signalInfo : TcoSignalInfo;
END_VAR
IF (_toWorkPos OR _moveWorkDefault.Busy) AND NOT inoDisableCondition THEN
    _signalInfo.GetSignalInfo(SIZEOF(inoDisableCondition), ADR(inoDisableCondition));
    Messenger.Warning(CONCAT('<#Movement suspended due to NOT#> : ', _signalInfo.SymbolPath));
    _toWorkPos := FALSE;

    IF (__ISVALIDREF(THIS^.inoToWorkPos)) THEN
        THIS^.inoToWorkPos := FALSE;
    END_IF;
END_IF
END_METHOD

END_FUNCTION_BLOCK
